RoboDK station: New Station (1).rdk

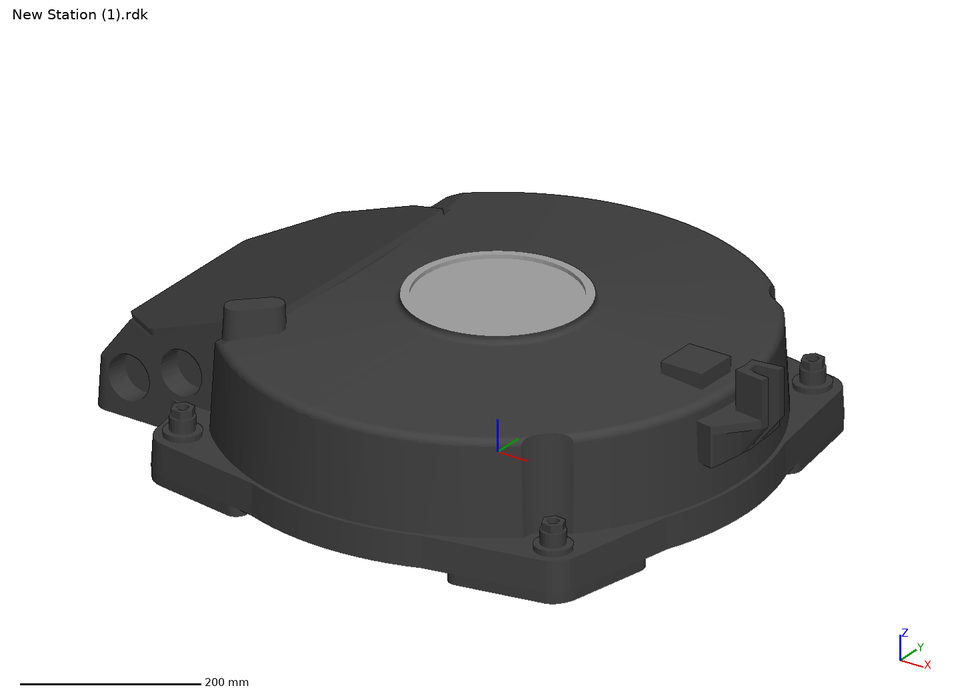
[picture v0: the station drawn from its stored meshes, robots at their saved joint values, targets as dots, program paths as lines]
Station New Station (1) (saved by RoboDK 5.7.4). Poses are relative to the parent item; angles as X-Y-Z fixed-axis rotations.
  - frame ABB IRB 580/12S Base at (0, 0, 0) mm
    - robot ABB IRB 580/12S: 6 axes, payload 12 kg, reach 2200 mm, repeatability 0.3 mm, weight 630 kg
        joint limits [-150, -70, -145, -360, -360, -720] to [150, 75, 145, 360, 360, 720]; home [0, 0, 0, 0, 0, 0]; saved at [0, 0, 0, 0, 0, 0]
